(* CoDeSys 2.3 export: F_WRITE_MAGIC_DOUBLE_CFG.EXP *)

(* POU FUN/PARAMETERS/F_WRITE_MAGIC_DOUBLE_CFG, ST *)
FUNCTION F_WRITE_MAGIC_DOUBLE_CFG : BOOL
VAR_INPUT
	sHead : STRING;
	wSize   :DWORD;
	pBuffer :POINTER TO BYTE;
END_VAR
VAR_IN_OUT
	wPos     : DWORD;
	stConfig : ST_MAGIC_DOUBLE_CFG;
END_VAR
VAR
END_VAR
F_ADD_STRINGX3_TO_BUFFER( S1:= '$n#', S2:= sHead, S3:=' - Parameters:$n', wSize := wSize, pBuffer := pBuffer, wPos := wPos );

F_ADD_STRINGX4_TO_BUFFER( S1:= CONCAT(sHead, '_P2Max' ), S2:='$t', S3:= REAL_TO_STRING( stConfig.P2Max ), S4:='$n', wSize := wSize, pBuffer := pBuffer, wPos := wPos );
F_ADD_STRINGX4_TO_BUFFER( S1:= CONCAT(sHead, '_P4Max' ), S2:='$t', S3:= REAL_TO_STRING( stConfig.P4Max ), S4:='$n', wSize := wSize, pBuffer := pBuffer, wPos := wPos );

F_ADD_STRINGX4_TO_BUFFER( S1:= CONCAT(sHead, '_EVPA4'   ), S2:='$t', S3:= INT_TO_STRING( stConfig.EVPA4  ), S4:='$n', wSize := wSize, pBuffer := pBuffer, wPos := wPos );
F_ADD_STRINGX4_TO_BUFFER( S1:= CONCAT(sHead, '_EVPA2'   ), S2:='$t', S3:= INT_TO_STRING( stConfig.EVPA2  ), S4:='$n', wSize := wSize, pBuffer := pBuffer, wPos := wPos );
F_ADD_STRINGX4_TO_BUFFER( S1:= CONCAT(sHead, '_EVPB4'   ), S2:='$t', S3:= INT_TO_STRING( stConfig.EVPB4  ), S4:='$n', wSize := wSize, pBuffer := pBuffer, wPos := wPos );
F_ADD_STRINGX4_TO_BUFFER( S1:= CONCAT(sHead, '_EVPB2'   ), S2:='$t', S3:= INT_TO_STRING( stConfig.EVPB2  ), S4:='$n', wSize := wSize, pBuffer := pBuffer, wPos := wPos );
F_ADD_STRINGX4_TO_BUFFER( S1:= CONCAT(sHead, '_EVPFA4'  ), S2:='$t', S3:= INT_TO_STRING( stConfig.EVPFA4 ), S4:='$n', wSize := wSize, pBuffer := pBuffer, wPos := wPos );
F_ADD_STRINGX4_TO_BUFFER( S1:= CONCAT(sHead, '_EVPFA2'  ), S2:='$t', S3:= INT_TO_STRING( stConfig.EVPFA2 ), S4:='$n', wSize := wSize, pBuffer := pBuffer, wPos := wPos );
F_ADD_STRINGX4_TO_BUFFER( S1:= CONCAT(sHead, '_EVPFB4'  ), S2:='$t', S3:= INT_TO_STRING( stConfig.EVPFB4 ), S4:='$n', wSize := wSize, pBuffer := pBuffer, wPos := wPos );
F_ADD_STRINGX4_TO_BUFFER( S1:= CONCAT(sHead, '_EVPFB2'  ), S2:='$t', S3:= INT_TO_STRING( stConfig.EVPFB2 ), S4:='$n', wSize := wSize, pBuffer := pBuffer, wPos := wPos );

F_ADD_STRINGX4_TO_BUFFER( S1:= CONCAT(sHead, '_EVPRA2'  ), S2:='$t', S3:= INT_TO_STRING( stConfig.EVPRA2  ), S4:='$n', wSize := wSize, pBuffer := pBuffer, wPos := wPos );

F_ADD_STRINGX4_TO_BUFFER( S1:= CONCAT(sHead, '_TgtLS4_In'  ), S2:='$t', S3:= REAL_TO_STRING( stConfig.TgtLS4_In  ), S4:='$n', wSize := wSize, pBuffer := pBuffer, wPos := wPos );
F_ADD_STRINGX4_TO_BUFFER( S1:= CONCAT(sHead, '_TgtLS4_Out' ), S2:='$t', S3:= REAL_TO_STRING( stConfig.TgtLS4_Out ), S4:='$n', wSize := wSize, pBuffer := pBuffer, wPos := wPos );
F_ADD_STRINGX4_TO_BUFFER( S1:= CONCAT(sHead, '_TgtLS2_In'  ), S2:='$t', S3:= REAL_TO_STRING( stConfig.TgtLS2_In  ), S4:='$n', wSize := wSize, pBuffer := pBuffer, wPos := wPos );
F_ADD_STRINGX4_TO_BUFFER( S1:= CONCAT(sHead, '_TgtLS2_Out' ), S2:='$t', S3:= REAL_TO_STRING( stConfig.TgtLS2_Out ), S4:='$n', wSize := wSize, pBuffer := pBuffer, wPos := wPos );

F_ADD_STRINGX4_TO_BUFFER( S1:= CONCAT(sHead, '_P_DB'     ), S2:='$t', S3:= REAL_TO_STRING( stConfig.P_DB     ), S4:='$n', wSize := wSize, pBuffer := pBuffer, wPos := wPos );
F_ADD_STRINGX4_TO_BUFFER( S1:= CONCAT(sHead, '_LS_DB'    ), S2:='$t', S3:= REAL_TO_STRING( stConfig.LS_DB    ), S4:='$n', wSize := wSize, pBuffer := pBuffer, wPos := wPos );

F_ADD_STRINGX4_TO_BUFFER( S1:= CONCAT(sHead, '_TimeMax'  ), S2:='$t', S3:= REAL_TO_STRING( stConfig.TimeMax  ), S4:='$n', wSize := wSize, pBuffer := pBuffer, wPos := wPos );
F_ADD_STRINGX4_TO_BUFFER( S1:= CONCAT(sHead, '_OutDelay' ), S2:='$t', S3:= REAL_TO_STRING( stConfig.OutDelay ), S4:='$n', wSize := wSize, pBuffer := pBuffer, wPos := wPos );
F_ADD_STRINGX4_TO_BUFFER( S1:= CONCAT(sHead, '_EVTDelay' ), S2:='$t', S3:= REAL_TO_STRING( stConfig.EVTDelay ), S4:='$n', wSize := wSize, pBuffer := pBuffer, wPos := wPos );

F_ADD_STRINGX4_TO_BUFFER( S1:= CONCAT(sHead, '_PP1'  ), S2:='$t', S3:= BOOL_TO_STRING( stConfig.PP1 ), S4:='$n', wSize := wSize, pBuffer := pBuffer, wPos := wPos );
F_ADD_STRINGX4_TO_BUFFER( S1:= CONCAT(sHead, '_PP2'  ), S2:='$t', S3:= BOOL_TO_STRING( stConfig.PP2 ), S4:='$n', wSize := wSize, pBuffer := pBuffer, wPos := wPos );
END_FUNCTION
